FUNCTION_BLOCK FB_RAT IMPLEMENTS I_Diverter
VAR_INPUT
    bSensorOccupied : BOOL;
    bSensorIsUp     : BOOL;
    bSensorIsDown   : BOOL;
END_VAR
VAR_OUTPUT
    bRatError          : BOOL;
    bIsLiftUp         : BOOL;
    bDivertMotorRun : BOOL;
END_VAR
VAR
    eRatState          : E_DiverterState := E_DiverterState.IDLE;
    fbLiftTimer     : TON;
    fbTravelTimer   : TON;
END_VAR

//fbLiftTimer(
//    IN := (eRatState = E_DiverterState.LIFTING OR eRatState = E_DiverterState.LOWERING),
//    PT := GVL_Config.T_RAT_LIFT_TIMEOUT
//);
//fbTravelTimer(IN := eRatState = E_DiverterState.DIVERTING, PT := T#6S);

IF fbLiftTimer.Q OR fbTravelTimer.Q THEN
    eRatState := E_DiverterState.FAULT;
END_IF

CASE eRatState OF
    E_DiverterState.IDLE:
        bIsLiftUp         := FALSE;
        bDivertMotorRun := FALSE;

    E_DiverterState.LIFTING:
        bIsLiftUp := TRUE;
        IF bSensorIsUp THEN
            eRatState := E_DiverterState.DIVERTING;
        END_IF

    E_DiverterState.DIVERTING:
        bIsLiftUp         := TRUE;
        bDivertMotorRun := TRUE;
        IF NOT bSensorOccupied THEN
            eRatState := E_DiverterState.LOWERING;
        END_IF

    E_DiverterState.LOWERING:
        bIsLiftUp         := FALSE;
        bDivertMotorRun := FALSE;
        IF bSensorIsDown THEN
            eRatState := E_DiverterState.DONE;
        END_IF
	
    E_DiverterState.FAULT:
        bIsLiftUp         := FALSE;
        bDivertMotorRun := FALSE;
        bRatError          := TRUE;
END_CASE

PROPERTY bError : BOOL
GET
bError := bRatError;
END_GET
END_PROPERTY

PROPERTY bLiftUp : BOOL
GET
bLiftUp := bIsLiftUp;
END_GET
END_PROPERTY

PROPERTY bTravelMotorRun : BOOL
GET
bTravelMotorRun := bDivertMotorRun;
END_GET
END_PROPERTY

PROPERTY eState : E_DiverterState
GET
eState := eRatState;
END_GET
END_PROPERTY

METHOD M_Divert
VAR_INPUT
END_VAR
IF eRatState = E_DiverterState.IDLE THEN
    eRatState := E_DiverterState.LIFTING;
END_IF
END_METHOD

METHOD M_Stop
VAR_INPUT
END_VAR
bIsLiftUp         := FALSE;
bDivertMotorRun := FALSE;
eRatState          := E_DiverterState.IDLE;
END_METHOD

END_FUNCTION_BLOCK

(* stored: Version 1.1.0.1, ProductVersion 3.1.4024.16
   POU FB_RAT: Id {a53e8369-ccc0-4a67-aaae-0302ede3efed}, SpecialFunc None
   Property bError: Id {bb000001-0000-0000-0000-000000000001}
   Get Get: Id {bb000002-0000-0000-0000-000000000001}
   Property bLiftUp: Id {bb000003-0000-0000-0000-000000000001}
   Get Get: Id {bb000004-0000-0000-0000-000000000001}
   Property bTravelMotorRun: Id {bb000005-0000-0000-0000-000000000001}
   Get Get: Id {bb000006-0000-0000-0000-000000000001}
   Property eState: Id {bb000007-0000-0000-0000-000000000001}
   Get Get: Id {bb000008-0000-0000-0000-000000000001}
   Method M_Divert: Id {bb000009-0000-0000-0000-000000000001}
   Method M_Stop: Id {bb000010-0000-0000-0000-000000000001} *)
